{attribute 'pack_mode' := '1'}
TYPE ST_ToggleSafetyCheck EXTENDS ST_MsgToPLC :
STRUCT
END_STRUCT
END_TYPE

(* stored: Version 1.1.0.1, ProductVersion 3.1.4024.3
   DUT ST_ToggleSafetyCheck: Id {e4b40c5e-58d8-40eb-9e15-83cd2581d5ba} *)
